// TIA Portal V20 export
DATA_BLOCK "Instance Equipment Modules"   // DB2
// stored: InstanceOfName FB Equipment Modules, InstanceOfType FB
"FB Equipment Modules"
   // VAR
   //    "Instance - Bas342" { S7_SetPoint := 'True'} : "FB - Bas342";
   //    "Instance - TableCheck - Process1" { S7_SetPoint := 'True'} : "FB - TableCheck";
   //    "Instance - TableCheck - Process2" { S7_SetPoint := 'True'} : "FB - TableCheck";
   //    "Instance - Sabload - P1 Left" { S7_SetPoint := 'True'} : "FB - Sabload";
   //    "Instance - Sabload - P1 Right" { S7_SetPoint := 'True'} : "FB - Sabload";
   //    "Instance - Sabload - P2 Left" { S7_SetPoint := 'True'} : "FB - Sabload";
   //    "Instance - Sabload - P2 Right" { S7_SetPoint := 'True'} : "FB - Sabload";
   // END_VAR
BEGIN
END_DATA_BLOCK
